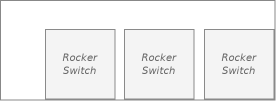
VISUALIZATION Visualization  // 276x101
    RockerSwitch (45,29 70x70), tooltip "'Transfer line 1'", variable: Visu.bStartTL1, behaviour: TOGGLE, style: Switch-RockerSwitch-Blue
    RockerSwitch (124,29 70x70), tooltip "'Transfer line 2'", variable: Visu.bStartTL2, behaviour: TOGGLE, style: Switch-RockerSwitch-Blue
    RockerSwitch (204,29 70x70), tooltip "'Transfer line 3'", variable: Visu.bStartTL3, behaviour: TOGGLE, style: Switch-RockerSwitch-Blue
END_VISUALIZATION

(* stored: Version 1.1.0.1, ProductVersion 3.1.4024.2
   Visu Visualization: Id {731c58f6-fc79-4ef3-9b0d-ec94f635715a} *)
